(* Logix 5000 project; controller CACLD_IR1_20200216 vendor 1 type 14 code 212 rev 32.11; software revision 32.00 *)

TASK MainTask (continuous, watchdog 500 ms) : MainProgram
TASK SafetyTask (periodic, rate 20 ms, priority 10, watchdog 20 ms, safety) : SafetyProgram

MODULES
   Local : vendor 1 type 14 code 212 (ICP 0, rev 32.11)
      R01_S05 : 1756-IA16 (ICP 5, rev 3.1, Input RPI 20 ms)
      R01_S07 : 1756-IB32 (ICP 7, rev 3.1, Input RPI 20 ms)
      R01_S06 : 1756-IB32 (ICP 6, rev 3.1, Input RPI 20 ms)
      R01_S08 : 1756-IB32 (ICP 8, rev 3.1, Input RPI 20 ms)
      R01_S09 : 1756-IB32 (ICP 9, rev 3.1, Input RPI 20 ms)
      R01_S10 : 1756-IB32 (ICP 10, rev 3.1, Input RPI 20 ms)
      R01_S11 : 1756-IB32 (ICP 11, rev 3.1, Input RPI 20 ms)
      R01_S12 : 1756-IB32 (ICP 12, rev 3.1, Input RPI 20 ms)
      R01_S13 : 1756-IB32 (ICP 13, rev 3.1, Input RPI 20 ms)
      R01_S014 : 1756-OB32 (ICP 14, rev 3.1, Output RPI 20 ms)
      R01_S015 : 1756-OB32 (ICP 15, rev 3.1, Output RPI 20 ms)
      DLR_S02 : vendor 1 type 12 code 200 (ICP 2, Ethernet 192.168.1.10, rev 11.1)
         MCP_R02 : 5094-AENTR (Ethernet 192.168.1.11, rev 3.1)
            MCP_R02_S01 : 5094-IB16S (5094 1, rev 1.1, SafetyInput RPI 20 ms, SafetyOutput RPI 20 ms)
            MCP_R02_S02 : 5094-OB16S (5094 2, rev 1.1, SafetyInput RPI 20 ms, SafetyOutput RPI 20 ms)
            MCP_R02_S03 : 5094-OB16S (5094 3, rev 1.1, SafetyInput RPI 20 ms, SafetyOutput RPI 20 ms)
            MCP_R02_S04 : 5094-OB16S (5094 4, rev 1.1, SafetyInput RPI 20 ms, SafetyOutput RPI 20 ms)
         RIO02_R01 : 5094-AENTR (Ethernet 192.168.1.13, rev 3.1)
            RIO02_R01_S02 : 5094-IB16 (5094 2, rev 1.1, StandardDataDriven RPI 5 ms)
            RIO02_R01_S01 : 5094-IB16 (5094 1, rev 1.1, StandardDataDriven RPI 5 ms)
            RIO02_R01_S03 : 5094-IB16 (5094 3, rev 1.1, StandardDataDriven RPI 5 ms)
            RIO02_R01_S04 : 5094-IB16 (5094 4, rev 1.1, StandardDataDriven RPI 5 ms)
            RIO02_R01_S05 : 5094-IB16 (5094 5, rev 1.1, StandardDataDriven RPI 5 ms)
            RIO02_R01_S07 : 5094-OB16S (5094 7, rev 1.1, SafetyOutput RPI 20 ms, SafetyInput RPI 20 ms)
            RIO02_R01_S06 : 5094-IB16S (5094 6, rev 1.1, SafetyOutput RPI 20 ms, SafetyInput RPI 20 ms)
         RIO01_R01 : 5094-AENTR (Ethernet 192.168.1.12, rev 3.1)
            RIO01_R01_S06 : 5094-IB16S (5094 6, rev 1.1, SafetyInput RPI 20 ms, SafetyOutput RPI 20 ms)
            RIO01_R01_S07 : 5094-OB16S (5094 7, rev 1.1, SafetyInput RPI 20 ms, SafetyOutput RPI 20 ms)
            RIO01_R01_S01 : 5094-IB16 (5094 1, rev 1.1, StandardDataDriven RPI 5 ms)
            RIO01_R01_S02 : 5094-IB16 (5094 2, rev 1.1, StandardDataDriven RPI 5 ms)
            RIO01_R01_S03 : 5094-IB16 (5094 3, rev 1.1, StandardDataDriven RPI 5 ms)
            RIO01_R01_S04 : 5094-IB16 (5094 4, rev 1.1, StandardDataDriven RPI 5 ms)
            RIO01_R01_S05 : 5094-IB16 (5094 5, rev 1.1, StandardDataDriven RPI 5 ms)
         RIO03_R01 : 5094-AENTR (Ethernet 192.168.1.14, rev 3.1)
            RIO03_R01_S02 : 5094-IB16 (5094 2, rev 1.1, StandardDataDriven RPI 5 ms)
            RIO03_R01_S01 : 5094-IB16 (5094 1, rev 1.1, StandardDataDriven RPI 5 ms)
            RIO03_R01_S03 : 5094-IB16 (5094 3, rev 1.1, StandardDataDriven RPI 5 ms)
            RIO03_R01_S04 : 5094-IB16 (5094 4, rev 1.1, StandardDataDriven RPI 5 ms)
            RIO03_R01_S05 : 5094-IB16 (5094 5, rev 1.1, StandardDataDriven RPI 5 ms)
            RIO03_R01_S07 : 5094-OB16S (5094 7, rev 1.1, SafetyInput RPI 20 ms, SafetyOutput RPI 20 ms)
            RIO03_R01_S06 : 5094-IB16S (5094 6, rev 1.1, SafetyInput RPI 20 ms, SafetyOutput RPI 20 ms)
         RIO04_R01 : 5094-AENTR (Ethernet 192.168.1.15, rev 3.1)
            RIO04_R01_S02 : 5094-IB16 (5094 2, rev 1.1, StandardDataDriven RPI 5 ms)
            RIO04_R01_S01 : 5094-IB16 (5094 1, rev 1.1, StandardDataDriven RPI 5 ms)
            RIO04_R01_S03 : 5094-IB16 (5094 3, rev 1.1, StandardDataDriven RPI 5 ms)
            RIO04_R01_S04 : 5094-IB16 (5094 4, rev 1.1, StandardDataDriven RPI 5 ms)
            RIO04_R01_S05 : 5094-IB16 (5094 5, rev 1.1, StandardDataDriven RPI 5 ms)
            RIO04_R01_S07 : 5094-OB16S (5094 7, rev 1.1, SafetyInput RPI 20 ms, SafetyOutput RPI 20 ms)
            RIO04_R01_S06 : 5094-IB16S (5094 6, rev 1.1, SafetyInput RPI 20 ms, SafetyOutput RPI 20 ms)
         RIO05_R01 : 5094-AENTR (Ethernet 192.168.1.16, rev 3.1)
            RIO05_R01_S02 : 5094-IB16 (5094 2, rev 1.1, StandardDataDriven RPI 5 ms)
            RIO05_R01_S01 : 5094-IB16 (5094 1, rev 1.1, StandardDataDriven RPI 5 ms)
            RIO05_R01_S03 : 5094-IB16 (5094 3, rev 1.1, StandardDataDriven RPI 5 ms)
            RIO05_R01_S04 : 5094-IB16 (5094 4, rev 1.1, StandardDataDriven RPI 5 ms)
            RIO05_R01_S05 : 5094-IB16 (5094 5, rev 1.1, StandardDataDriven RPI 5 ms)
            RIO05_R01_S07 : 5094-OB16S (5094 7, rev 1.1, SafetyInput RPI 20 ms, SafetyOutput RPI 20 ms)
            RIO05_R01_S06 : 5094-IB16S (5094 6, rev 1.1, SafetyInput RPI 20 ms, SafetyOutput RPI 20 ms)
      DLR_S04 : vendor 1 type 12 code 200 (ICP 4, Ethernet 192.168.1.10, rev 11.1)
         RIO06_R01 : 5094-AENTR (Ethernet 192.168.1.11, rev 3.1)
            RIO06_R01_S07 : 5094-OB16S (5094 7, rev 1.1, SafetyInput RPI 20 ms, SafetyOutput RPI 20 ms)
            RIO06_R01_S01 : 5094-IB16 (5094 1, rev 1.1, StandardDataDriven RPI 5 ms)
            RIO06_R01_S02 : 5094-IB16 (5094 2, rev 1.1, StandardDataDriven RPI 5 ms)
            RIO06_R01_S03 : 5094-IB16 (5094 3, rev 1.1, StandardDataDriven RPI 5 ms)
            RIO06_R01_S04 : 5094-IB16 (5094 4, rev 1.1, StandardDataDriven RPI 5 ms)
            RIO06_R01_S06 : 5094-IB16S (5094 6, rev 1.1, SafetyInput RPI 20 ms, SafetyOutput RPI 20 ms)
            RIO06_R01_S05 : 5094-IB16 (5094 5, rev 1.1, StandardDataDriven RPI 5 ms)
         RIO07_R01 : 5094-AENTR (Ethernet 192.168.1.12, rev 3.1)
            RIO07_R01_S02 : 5094-IB16 (5094 2, rev 1.1, StandardDataDriven RPI 5 ms)
            RIO07_R01_S01 : 5094-IB16 (5094 1, rev 1.1, StandardDataDriven RPI 5 ms)
            RIO07_R01_S03 : 5094-IB16 (5094 3, rev 1.1, StandardDataDriven RPI 5 ms)
            RIO07_R01_S04 : 5094-IB16 (5094 4, rev 1.1, StandardDataDriven RPI 5 ms)
            RIO07_R01_S05 : 5094-IB16 (5094 5, rev 1.1, StandardDataDriven RPI 5 ms)
            RIO07_R01_S07 : 5094-OB16S (5094 7, rev 1.1, SafetyInput RPI 20 ms, SafetyOutput RPI 20 ms)
            RIO07_R01_S06 : 5094-IB16S (5094 6, rev 1.1, SafetyInput RPI 20 ms, SafetyOutput RPI 20 ms)
         RIO08_R01 : 5094-AENTR (Ethernet 192.168.1.13, rev 3.1)
            RIO08_R01_S02 : 5094-IB16 (5094 2, rev 1.1, StandardDataDriven RPI 5 ms)
            RIO08_R01_S01 : 5094-IB16 (5094 1, rev 1.1, StandardDataDriven RPI 5 ms)
            RIO08_R01_S03 : 5094-IB16 (5094 3, rev 1.1, StandardDataDriven RPI 5 ms)
            RIO08_R01_S04 : 5094-IB16 (5094 4, rev 1.1, StandardDataDriven RPI 5 ms)
            RIO08_R01_S05 : 5094-IB16 (5094 5, rev 1.1, StandardDataDriven RPI 5 ms)
            RIO08_R01_S07 : 5094-OB16S (5094 7, rev 1.1, SafetyInput RPI 20 ms, SafetyOutput RPI 20 ms)
            RIO08_R01_S06 : 5094-IB16S (5094 6, rev 1.1, SafetyInput RPI 20 ms, SafetyOutput RPI 20 ms)
END_MODULES

PROGRAM MainProgram   (* main routine MainRoutine *)

ROUTINE MainRoutine   (* ladder *)
END_ROUTINE
END_PROGRAM

PROGRAM SafetyProgram   (* main routine MainRoutine, safety *)

ROUTINE MainRoutine   (* ladder *)
END_ROUTINE
END_PROGRAM
